// TIA Portal V15.1 export
// export: Created 2024-05-17T05:38:58.758149Z, ExportSetting WithDefaults, DisplayName Totally Integrated Automation Portal, DisplayVersion V15.1 Update 5, DisplayName TIA Portal Openness, DisplayVersion V15.1 Update 5, DisplayName SINAMICS Startdrive Advanced, DisplayVersion V15.1, DisplayName G130, G150, S120, S150, SINAMICS MV, S210, DisplayVersion V15.1, DisplayName G110M, G120, G120C, G120D, G120P, DisplayVersion V15.1, DisplayName STEP 7 Professional, DisplayVersion V15.1 Update 5, DisplayName STEP 7 Safety, DisplayVersion V15.1, DisplayName WinCC Professional, DisplayVersion V15.1 Update 5, DisplayName SIMATIC Visualization Architect, DisplayVersion V15.1
FUNCTION "209230ZS01PNIODiag" : Void   // FC424, FBD
TITLE = 209230ZS01PNIODiag
{ S7_Optimized_Access := 'FALSE' }
AUTHOR : JS
NAME : Mot001
VERSION : 0.1
// stored: AutoNumber false, IsIECCheckEnabled false, SetENOAutomatically False, UDAEnableTagReadback false
   VAR_OUTPUT
      O_AlarmA : Bool;   // Alarm A
      O_AlarmB : Bool;   // Alarm B
      O_AlarmC : Bool;   // Alarm C
      O_AlarmD : Bool;   // Alarm D
      O_AlarmABCondition : Bool;   // Alarms resetable
      H_IAnim : Word;   // Animation bits to Icon in WinCC
   END_VAR
   VAR_TEMP   // added for the SCL form of the ladder/FBD networks
      _w1 : Bool;
   END_VAR
BEGIN

REGION Network 1: **** --------------------- ET200sp I/O --------------------- ****
END_REGION

REGION Network 2: **** 3 - Communication - Devices **** 209230AS10-JW60 - ET200sp I/O - Busnode 230AS10 - node 60
   // Profinet device don't exist - ET200sp I/O - Busnode 230AS10 - node 60
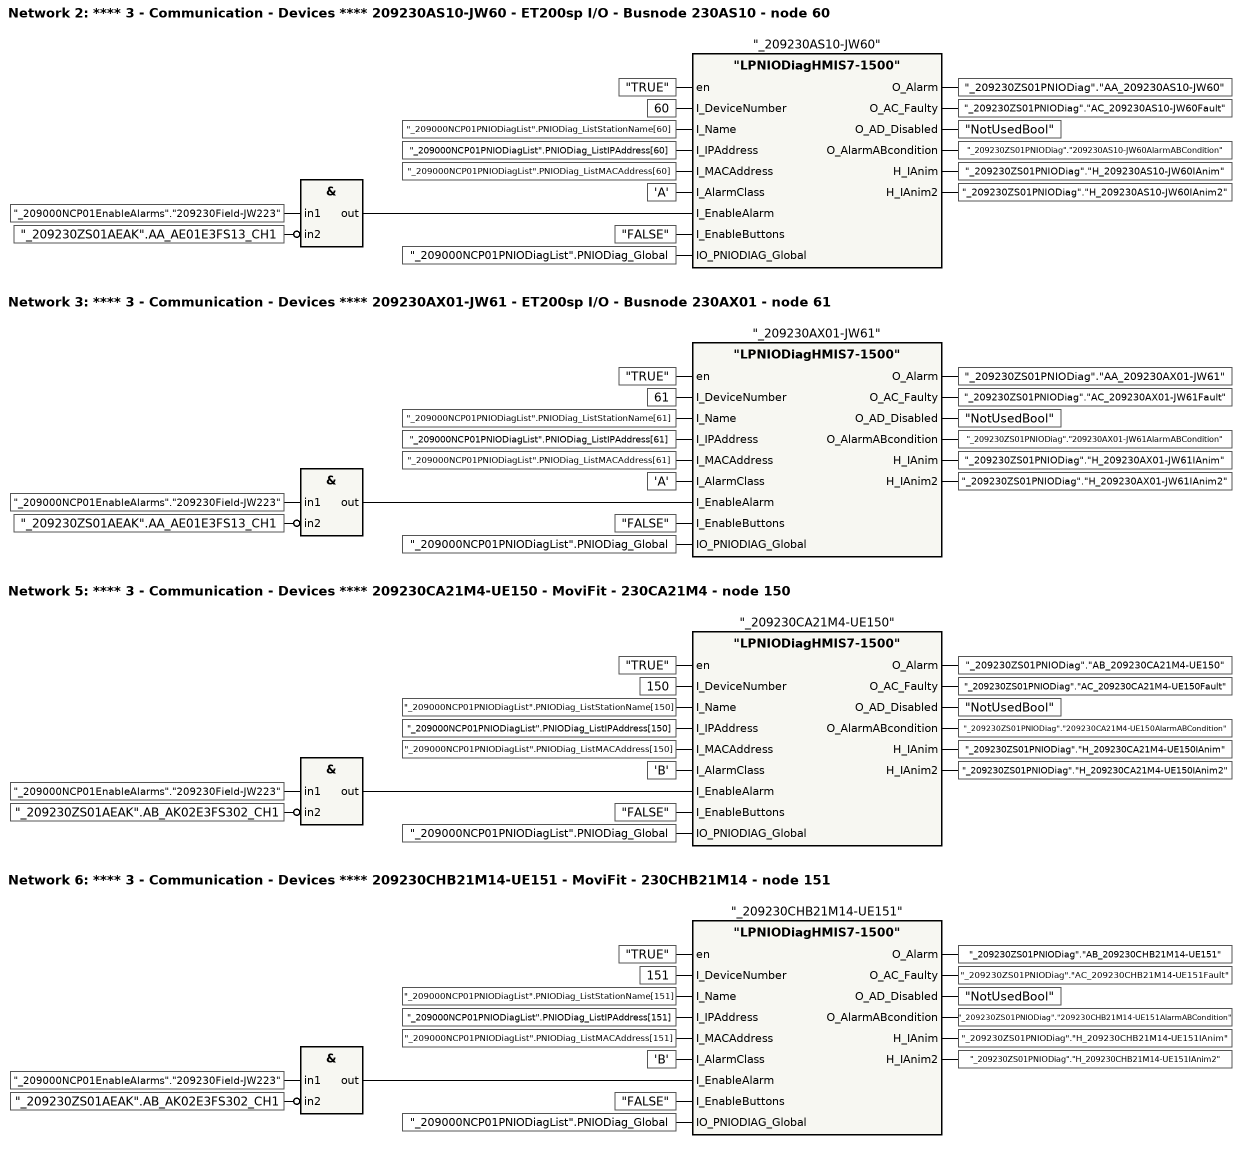
   IF "TRUE" THEN
       "_209230AS10-JW60"(I_DeviceNumber := 60,   // "LPNIODiagHMIS7-1500"
                          I_Name := "_209000NCP01PNIODiagList".PNIODiag_ListStationName[60],
                          I_IPAddress := "_209000NCP01PNIODiagList".PNIODiag_ListIPAddress[60],
                          I_MACAddress := "_209000NCP01PNIODiagList".PNIODiag_ListMACAddress[60],
                          I_AlarmClass := 'A',
                          I_EnableAlarm := "_209000NCP01EnableAlarms"."209230Field-JW223" AND NOT "_209230ZS01AEAK".AA_AE01E3FS13_CH1,
                          I_EnableButtons := "FALSE",
                          IO_PNIODIAG_Global := "_209000NCP01PNIODiagList".PNIODiag_Global,
                          O_Alarm => "_209230ZS01PNIODiag"."AA_209230AS10-JW60",
                          O_AC_Faulty => "_209230ZS01PNIODiag"."AC_209230AS10-JW60Fault",
                          O_AD_Disabled => "NotUsedBool",
                          O_AlarmABcondition => "_209230ZS01PNIODiag"."209230AS10-JW60AlarmABCondition",
                          H_IAnim => "_209230ZS01PNIODiag"."H_209230AS10-JW60IAnim",
                          H_IAnim2 => "_209230ZS01PNIODiag"."H_209230AS10-JW60IAnim2");
   END_IF;
END_REGION

REGION Network 3: **** 3 - Communication - Devices **** 209230AX01-JW61 - ET200sp I/O - Busnode 230AX01 - node 61
   // Profinet device don't exist - ET200sp I/O - Busnode 230AX01 - node 61
   IF "TRUE" THEN
       "_209230AX01-JW61"(I_DeviceNumber := 61,   // "LPNIODiagHMIS7-1500"
                          I_Name := "_209000NCP01PNIODiagList".PNIODiag_ListStationName[61],
                          I_IPAddress := "_209000NCP01PNIODiagList".PNIODiag_ListIPAddress[61],
                          I_MACAddress := "_209000NCP01PNIODiagList".PNIODiag_ListMACAddress[61],
                          I_AlarmClass := 'A',
                          I_EnableAlarm := "_209000NCP01EnableAlarms"."209230Field-JW223" AND NOT "_209230ZS01AEAK".AA_AE01E3FS13_CH1,
                          I_EnableButtons := "FALSE",
                          IO_PNIODIAG_Global := "_209000NCP01PNIODiagList".PNIODiag_Global,
                          O_Alarm => "_209230ZS01PNIODiag"."AA_209230AX01-JW61",
                          O_AC_Faulty => "_209230ZS01PNIODiag"."AC_209230AX01-JW61Fault",
                          O_AD_Disabled => "NotUsedBool",
                          O_AlarmABcondition => "_209230ZS01PNIODiag"."209230AX01-JW61AlarmABCondition",
                          H_IAnim => "_209230ZS01PNIODiag"."H_209230AX01-JW61IAnim",
                          H_IAnim2 => "_209230ZS01PNIODiag"."H_209230AX01-JW61IAnim2");
   END_IF;
END_REGION

REGION Network 4: **** --------------------- Drive --------------------- ****
END_REGION

REGION Network 5: **** 3 - Communication - Devices **** 209230CA21M4-UE150 - MoviFit - 230CA21M4 - node 150
   // Profinet device don't exist - MoviFit - 230CA21M4 - node 150
   IF "TRUE" THEN
       "_209230CA21M4-UE150"(I_DeviceNumber := 150,   // "LPNIODiagHMIS7-1500"
                             I_Name := "_209000NCP01PNIODiagList".PNIODiag_ListStationName[150],
                             I_IPAddress := "_209000NCP01PNIODiagList".PNIODiag_ListIPAddress[150],
                             I_MACAddress := "_209000NCP01PNIODiagList".PNIODiag_ListMACAddress[150],
                             I_AlarmClass := 'B',
                             I_EnableAlarm := "_209000NCP01EnableAlarms"."209230Field-JW223" AND NOT "_209230ZS01AEAK".AB_AK02E3FS302_CH1,
                             I_EnableButtons := "FALSE",
                             IO_PNIODIAG_Global := "_209000NCP01PNIODiagList".PNIODiag_Global,
                             O_Alarm => "_209230ZS01PNIODiag"."AB_209230CA21M4-UE150",
                             O_AC_Faulty => "_209230ZS01PNIODiag"."AC_209230CA21M4-UE150Fault",
                             O_AD_Disabled => "NotUsedBool",
                             O_AlarmABcondition => "_209230ZS01PNIODiag"."209230CA21M4-UE150AlarmABCondition",
                             H_IAnim => "_209230ZS01PNIODiag"."H_209230CA21M4-UE150IAnim",
                             H_IAnim2 => "_209230ZS01PNIODiag"."H_209230CA21M4-UE150IAnim2");
   END_IF;
END_REGION

REGION Network 6: **** 3 - Communication - Devices **** 209230CHB21M14-UE151 - MoviFit - 230CHB21M14 - node 151
   // Profinet device don't exist - MoviFit - 230CHB21M14 - node 151
   IF "TRUE" THEN
       "_209230CHB21M14-UE151"(I_DeviceNumber := 151,   // "LPNIODiagHMIS7-1500"
                               I_Name := "_209000NCP01PNIODiagList".PNIODiag_ListStationName[151],
                               I_IPAddress := "_209000NCP01PNIODiagList".PNIODiag_ListIPAddress[151],
                               I_MACAddress := "_209000NCP01PNIODiagList".PNIODiag_ListMACAddress[151],
                               I_AlarmClass := 'B',
                               I_EnableAlarm := "_209000NCP01EnableAlarms"."209230Field-JW223" AND NOT "_209230ZS01AEAK".AB_AK02E3FS302_CH1,
                               I_EnableButtons := "FALSE",
                               IO_PNIODIAG_Global := "_209000NCP01PNIODiagList".PNIODiag_Global,
                               O_Alarm => "_209230ZS01PNIODiag"."AB_209230CHB21M14-UE151",
                               O_AC_Faulty => "_209230ZS01PNIODiag"."AC_209230CHB21M14-UE151Fault",
                               O_AD_Disabled => "NotUsedBool",
                               O_AlarmABcondition => "_209230ZS01PNIODiag"."209230CHB21M14-UE151AlarmABCondition",
                               H_IAnim => "_209230ZS01PNIODiag"."H_209230CHB21M14-UE151IAnim",
                               H_IAnim2 => "_209230ZS01PNIODiag"."H_209230CHB21M14-UE151IAnim2");
   END_IF;
END_REGION

REGION Network 7: **** 3 - Communication - Devices **** 209230CHB22M14-UE152 - MoviFit - 230CHB22M14 - node 152
   // Profinet device don't exist - MoviFit - 230CHB22M14 - node 152
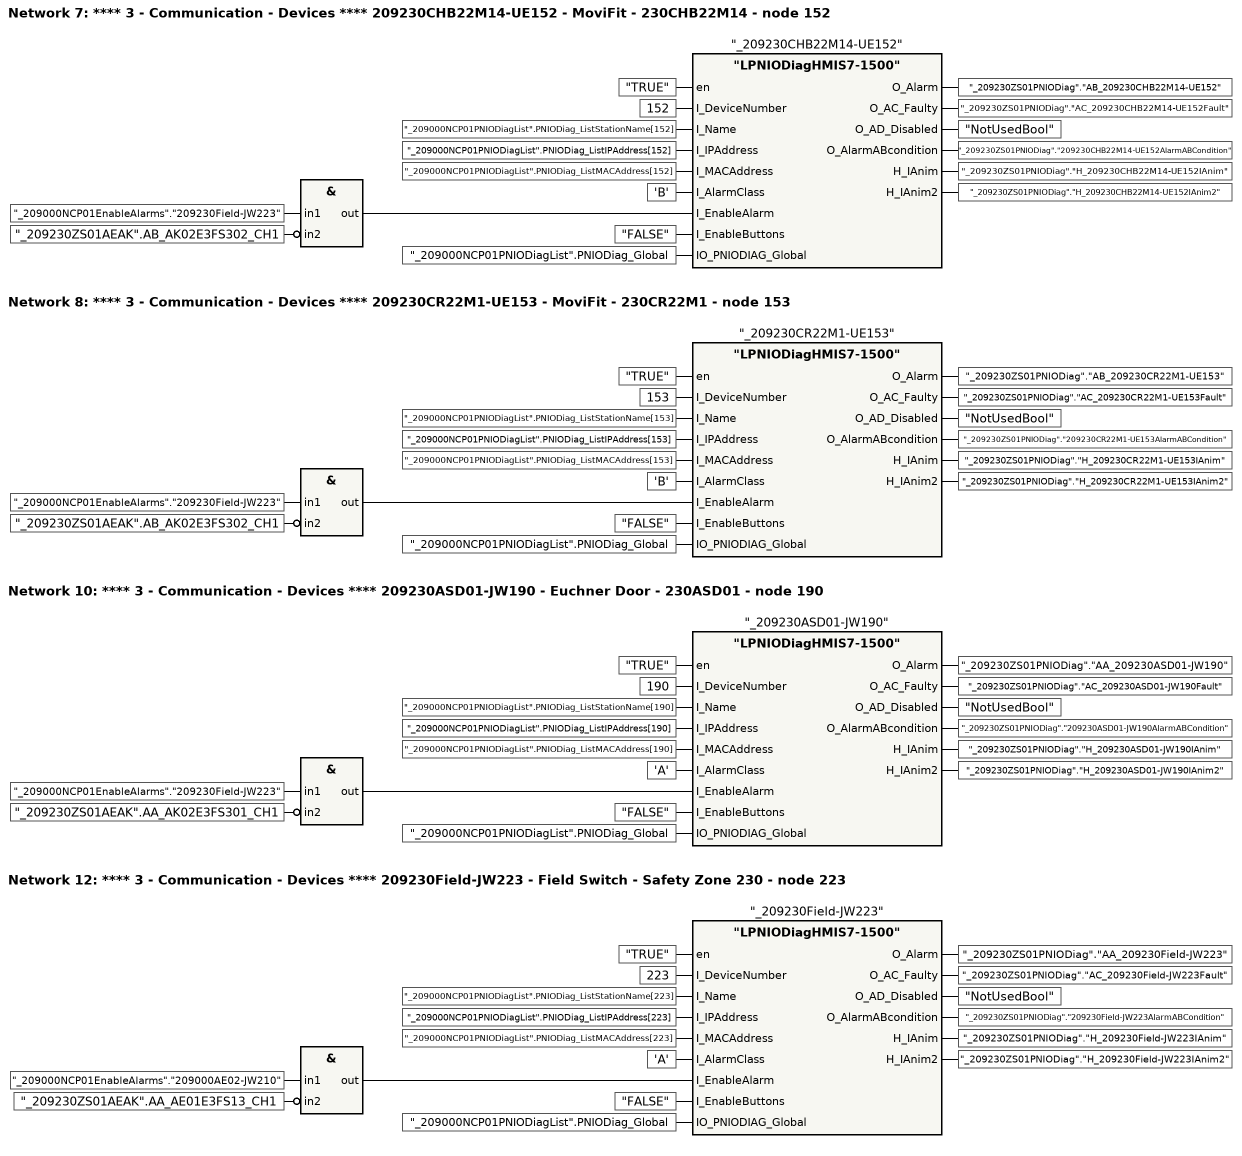
   IF "TRUE" THEN
       "_209230CHB22M14-UE152"(I_DeviceNumber := 152,   // "LPNIODiagHMIS7-1500"
                               I_Name := "_209000NCP01PNIODiagList".PNIODiag_ListStationName[152],
                               I_IPAddress := "_209000NCP01PNIODiagList".PNIODiag_ListIPAddress[152],
                               I_MACAddress := "_209000NCP01PNIODiagList".PNIODiag_ListMACAddress[152],
                               I_AlarmClass := 'B',
                               I_EnableAlarm := "_209000NCP01EnableAlarms"."209230Field-JW223" AND NOT "_209230ZS01AEAK".AB_AK02E3FS302_CH1,
                               I_EnableButtons := "FALSE",
                               IO_PNIODIAG_Global := "_209000NCP01PNIODiagList".PNIODiag_Global,
                               O_Alarm => "_209230ZS01PNIODiag"."AB_209230CHB22M14-UE152",
                               O_AC_Faulty => "_209230ZS01PNIODiag"."AC_209230CHB22M14-UE152Fault",
                               O_AD_Disabled => "NotUsedBool",
                               O_AlarmABcondition => "_209230ZS01PNIODiag"."209230CHB22M14-UE152AlarmABCondition",
                               H_IAnim => "_209230ZS01PNIODiag"."H_209230CHB22M14-UE152IAnim",
                               H_IAnim2 => "_209230ZS01PNIODiag"."H_209230CHB22M14-UE152IAnim2");
   END_IF;
END_REGION

REGION Network 8: **** 3 - Communication - Devices **** 209230CR22M1-UE153 - MoviFit - 230CR22M1 - node 153
   // Profinet device don't exist - MoviFit - 230CR22M1 - node 153
   IF "TRUE" THEN
       "_209230CR22M1-UE153"(I_DeviceNumber := 153,   // "LPNIODiagHMIS7-1500"
                             I_Name := "_209000NCP01PNIODiagList".PNIODiag_ListStationName[153],
                             I_IPAddress := "_209000NCP01PNIODiagList".PNIODiag_ListIPAddress[153],
                             I_MACAddress := "_209000NCP01PNIODiagList".PNIODiag_ListMACAddress[153],
                             I_AlarmClass := 'B',
                             I_EnableAlarm := "_209000NCP01EnableAlarms"."209230Field-JW223" AND NOT "_209230ZS01AEAK".AB_AK02E3FS302_CH1,
                             I_EnableButtons := "FALSE",
                             IO_PNIODIAG_Global := "_209000NCP01PNIODiagList".PNIODiag_Global,
                             O_Alarm => "_209230ZS01PNIODiag"."AB_209230CR22M1-UE153",
                             O_AC_Faulty => "_209230ZS01PNIODiag"."AC_209230CR22M1-UE153Fault",
                             O_AD_Disabled => "NotUsedBool",
                             O_AlarmABcondition => "_209230ZS01PNIODiag"."209230CR22M1-UE153AlarmABCondition",
                             H_IAnim => "_209230ZS01PNIODiag"."H_209230CR22M1-UE153IAnim",
                             H_IAnim2 => "_209230ZS01PNIODiag"."H_209230CR22M1-UE153IAnim2");
   END_IF;
END_REGION

REGION Network 9: **** --------------------- Euchner Door --------------------- ****
END_REGION

REGION Network 10: **** 3 - Communication - Devices **** 209230ASD01-JW190 - Euchner Door - 230ASD01 - node 190
   // Profinet device don't exist - Euchner Door - 230ASD01 - node 190
   IF "TRUE" THEN
       "_209230ASD01-JW190"(I_DeviceNumber := 190,   // "LPNIODiagHMIS7-1500"
                            I_Name := "_209000NCP01PNIODiagList".PNIODiag_ListStationName[190],
                            I_IPAddress := "_209000NCP01PNIODiagList".PNIODiag_ListIPAddress[190],
                            I_MACAddress := "_209000NCP01PNIODiagList".PNIODiag_ListMACAddress[190],
                            I_AlarmClass := 'A',
                            I_EnableAlarm := "_209000NCP01EnableAlarms"."209230Field-JW223" AND NOT "_209230ZS01AEAK".AA_AK02E3FS301_CH1,
                            I_EnableButtons := "FALSE",
                            IO_PNIODIAG_Global := "_209000NCP01PNIODiagList".PNIODiag_Global,
                            O_Alarm => "_209230ZS01PNIODiag"."AA_209230ASD01-JW190",
                            O_AC_Faulty => "_209230ZS01PNIODiag"."AC_209230ASD01-JW190Fault",
                            O_AD_Disabled => "NotUsedBool",
                            O_AlarmABcondition => "_209230ZS01PNIODiag"."209230ASD01-JW190AlarmABCondition",
                            H_IAnim => "_209230ZS01PNIODiag"."H_209230ASD01-JW190IAnim",
                            H_IAnim2 => "_209230ZS01PNIODiag"."H_209230ASD01-JW190IAnim2");
   END_IF;
END_REGION

REGION Network 11: **** --------------------- Field Switch --------------------- ****
END_REGION

REGION Network 12: **** 3 - Communication - Devices **** 209230Field-JW223 - Field Switch - Safety Zone 230 - node 223
   // Profinet device don't exist - Field Switch - Safety Zone 230 - node 223
   IF "TRUE" THEN
       "_209230Field-JW223"(I_DeviceNumber := 223,   // "LPNIODiagHMIS7-1500"
                            I_Name := "_209000NCP01PNIODiagList".PNIODiag_ListStationName[223],
                            I_IPAddress := "_209000NCP01PNIODiagList".PNIODiag_ListIPAddress[223],
                            I_MACAddress := "_209000NCP01PNIODiagList".PNIODiag_ListMACAddress[223],
                            I_AlarmClass := 'A',
                            I_EnableAlarm := "_209000NCP01EnableAlarms"."209000AE02-JW210" AND NOT "_209230ZS01AEAK".AA_AE01E3FS13_CH1,
                            I_EnableButtons := "FALSE",
                            IO_PNIODIAG_Global := "_209000NCP01PNIODiagList".PNIODiag_Global,
                            O_Alarm => "_209230ZS01PNIODiag"."AA_209230Field-JW223",
                            O_AC_Faulty => "_209230ZS01PNIODiag"."AC_209230Field-JW223Fault",
                            O_AD_Disabled => "NotUsedBool",
                            O_AlarmABcondition => "_209230ZS01PNIODiag"."209230Field-JW223AlarmABCondition",
                            H_IAnim => "_209230ZS01PNIODiag"."H_209230Field-JW223IAnim",
                            H_IAnim2 => "_209230ZS01PNIODiag"."H_209230Field-JW223IAnim2");
   END_IF;
END_REGION

REGION Network 13: **** -------------------------------------------------- ****
END_REGION

REGION Network 14: **** 4.6 - Machine Status - Indications **** Icon animation
   // Icon animation
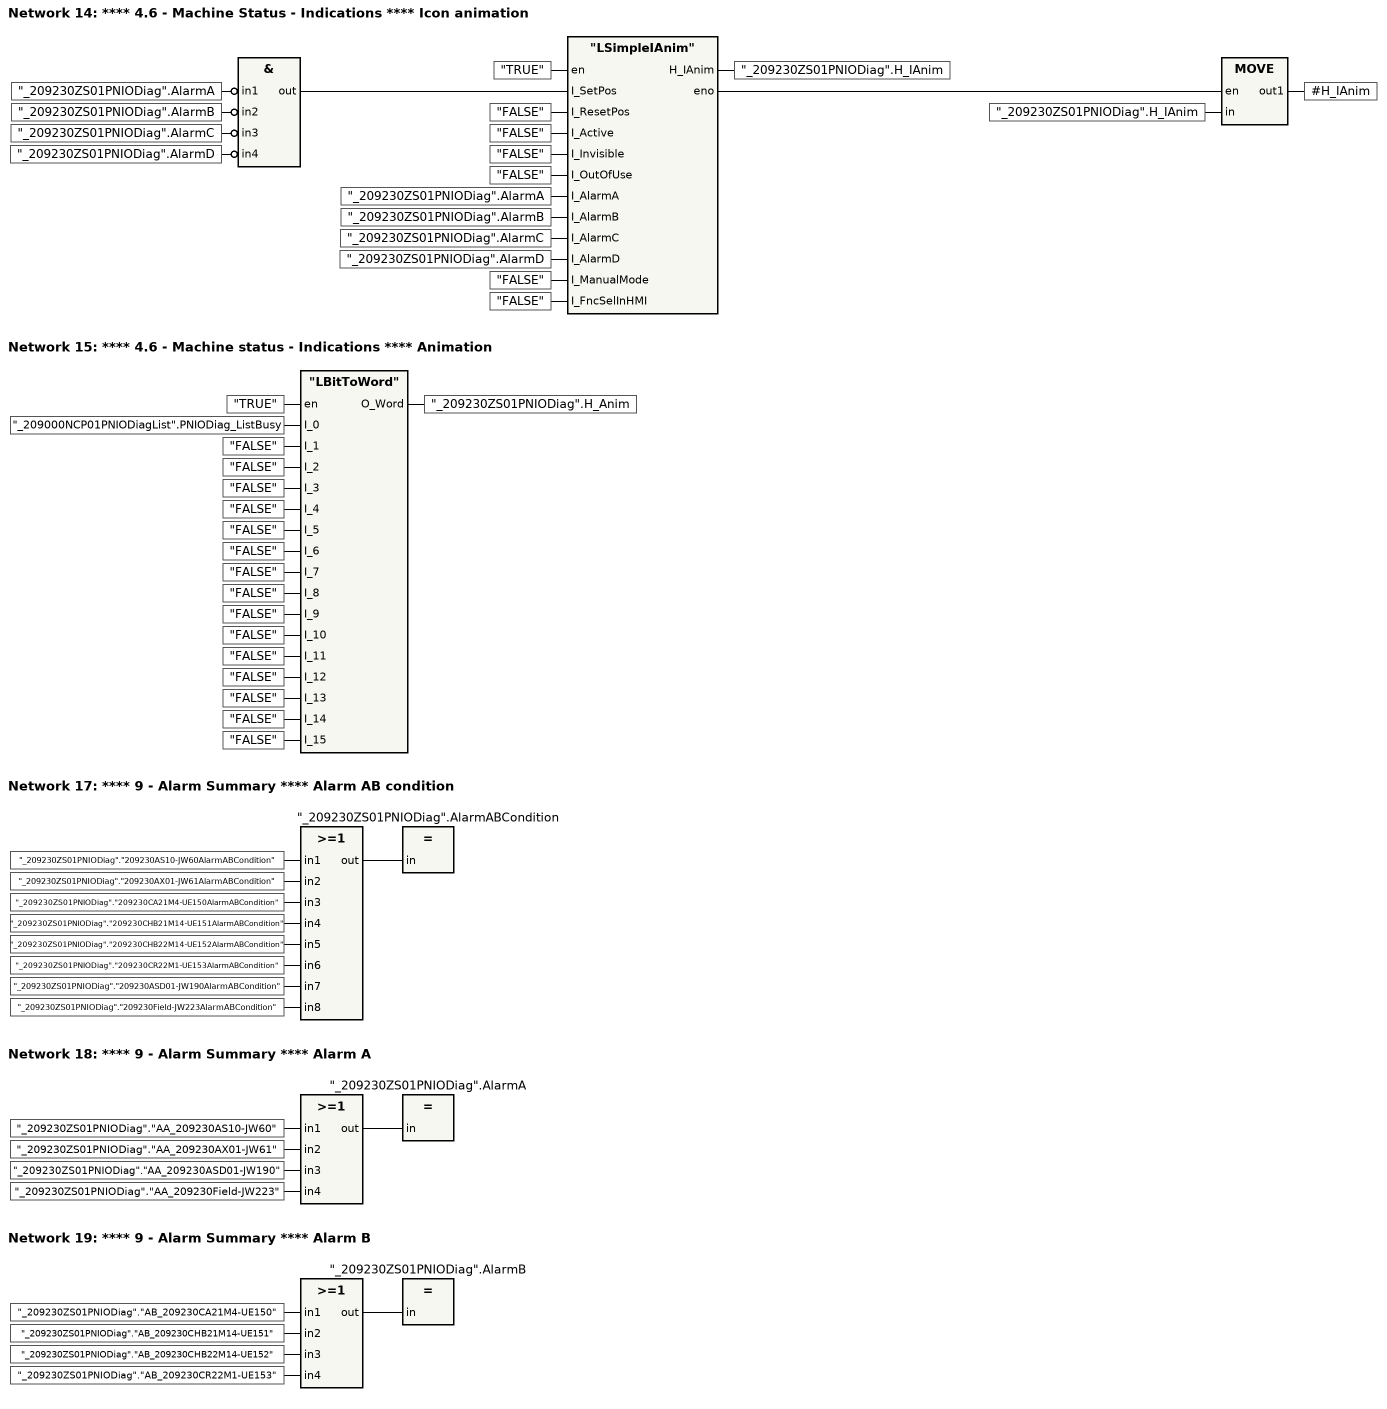
   "LSimpleIAnim"(EN := "TRUE",
                  I_SetPos := NOT "_209230ZS01PNIODiag".AlarmA AND NOT "_209230ZS01PNIODiag".AlarmB AND NOT "_209230ZS01PNIODiag".AlarmC AND NOT "_209230ZS01PNIODiag".AlarmD,
                  I_ResetPos := "FALSE",
                  I_Active := "FALSE",
                  I_Invisible := "FALSE",
                  I_OutOfUse := "FALSE",
                  I_AlarmA := "_209230ZS01PNIODiag".AlarmA,
                  I_AlarmB := "_209230ZS01PNIODiag".AlarmB,
                  I_AlarmC := "_209230ZS01PNIODiag".AlarmC,
                  I_AlarmD := "_209230ZS01PNIODiag".AlarmD,
                  I_ManualMode := "FALSE",
                  I_FncSelInHMI := "FALSE",
                  H_IAnim => "_209230ZS01PNIODiag".H_IAnim,
                  ENO => #_w1);
   IF #_w1 THEN #H_IAnim := "_209230ZS01PNIODiag".H_IAnim; END_IF;
END_REGION

REGION Network 15: **** 4.6 - Machine status - Indications **** Animation
   // Animation
   IF "TRUE" THEN
       "LBitToWord"(I_0 := "_209000NCP01PNIODiagList".PNIODiag_ListBusy,
                    I_1 := "FALSE",
                    I_2 := "FALSE",
                    I_3 := "FALSE",
                    I_4 := "FALSE",
                    I_5 := "FALSE",
                    I_6 := "FALSE",
                    I_7 := "FALSE",
                    I_8 := "FALSE",
                    I_9 := "FALSE",
                    I_10 := "FALSE",
                    I_11 := "FALSE",
                    I_12 := "FALSE",
                    I_13 := "FALSE",
                    I_14 := "FALSE",
                    I_15 := "FALSE",
                    O_Word => "_209230ZS01PNIODiag".H_Anim);
   END_IF;
END_REGION

NETWORK
TITLE = **** 4.6 - Machine Status - Indications **** Animation DB number
// DB number
      OPN   "_209230ZS01PNIODiag";
      L     DBNO;
      T     "_209230ZS01PNIODiag".H_DBnr;

REGION Network 17: **** 9 - Alarm Summary **** Alarm AB condition
   // Summary of Alarm AB condition
   "_209230ZS01PNIODiag".AlarmABCondition := "_209230ZS01PNIODiag"."209230AS10-JW60AlarmABCondition" OR "_209230ZS01PNIODiag"."209230AX01-JW61AlarmABCondition" OR "_209230ZS01PNIODiag"."209230CA21M4-UE150AlarmABCondition" OR "_209230ZS01PNIODiag"."209230CHB21M14-UE151AlarmABCondition" OR "_209230ZS01PNIODiag"."209230CHB22M14-UE152AlarmABCondition" OR "_209230ZS01PNIODiag"."209230CR22M1-UE153AlarmABCondition" OR "_209230ZS01PNIODiag"."209230ASD01-JW190AlarmABCondition" OR "_209230ZS01PNIODiag"."209230Field-JW223AlarmABCondition";
END_REGION

REGION Network 18: **** 9 - Alarm Summary **** Alarm A
   // Summary of alarms A
   "_209230ZS01PNIODiag".AlarmA := "_209230ZS01PNIODiag"."AA_209230AS10-JW60" OR "_209230ZS01PNIODiag"."AA_209230AX01-JW61" OR "_209230ZS01PNIODiag"."AA_209230ASD01-JW190" OR "_209230ZS01PNIODiag"."AA_209230Field-JW223";
END_REGION

REGION Network 19: **** 9 - Alarm Summary **** Alarm B
   // Summary of alarms B
   "_209230ZS01PNIODiag".AlarmB := "_209230ZS01PNIODiag"."AB_209230CA21M4-UE150" OR "_209230ZS01PNIODiag"."AB_209230CHB21M14-UE151" OR "_209230ZS01PNIODiag"."AB_209230CHB22M14-UE152" OR "_209230ZS01PNIODiag"."AB_209230CR22M1-UE153";
END_REGION

REGION Network 20: **** 9 - Alarm Summary **** Alarm C
   // Summary of alarms C
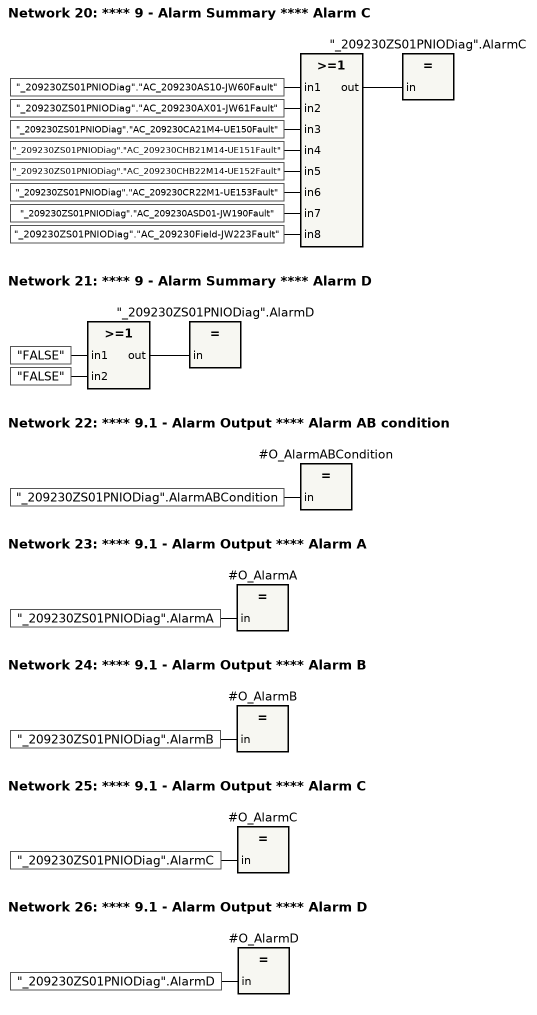
   "_209230ZS01PNIODiag".AlarmC := "_209230ZS01PNIODiag"."AC_209230AS10-JW60Fault" OR "_209230ZS01PNIODiag"."AC_209230AX01-JW61Fault" OR "_209230ZS01PNIODiag"."AC_209230CA21M4-UE150Fault" OR "_209230ZS01PNIODiag"."AC_209230CHB21M14-UE151Fault" OR "_209230ZS01PNIODiag"."AC_209230CHB22M14-UE152Fault" OR "_209230ZS01PNIODiag"."AC_209230CR22M1-UE153Fault" OR "_209230ZS01PNIODiag"."AC_209230ASD01-JW190Fault" OR "_209230ZS01PNIODiag"."AC_209230Field-JW223Fault";
END_REGION

REGION Network 21: **** 9 - Alarm Summary **** Alarm D
   // Summary of alarms D
   "_209230ZS01PNIODiag".AlarmD := "FALSE" OR "FALSE";
END_REGION

REGION Network 22: **** 9.1 - Alarm Output **** Alarm AB condition
   // Alarm AB condition
   #O_AlarmABCondition := "_209230ZS01PNIODiag".AlarmABCondition;
END_REGION

REGION Network 23: **** 9.1 - Alarm Output **** Alarm A
   // Output Alarm A
   #O_AlarmA := "_209230ZS01PNIODiag".AlarmA;
END_REGION

REGION Network 24: **** 9.1 - Alarm Output **** Alarm B
   // Output Alarm B
   #O_AlarmB := "_209230ZS01PNIODiag".AlarmB;
END_REGION

REGION Network 25: **** 9.1 - Alarm Output **** Alarm C
   // Output Alarm A
   #O_AlarmC := "_209230ZS01PNIODiag".AlarmC;
END_REGION

REGION Network 26: **** 9.1 - Alarm Output **** Alarm D
   // Output Alarm D
   #O_AlarmD := "_209230ZS01PNIODiag".AlarmD;
END_REGION

REGION Network 27: **** 9.2 - Alarm DWord**** Alarm To DWord
   // Alarm Word
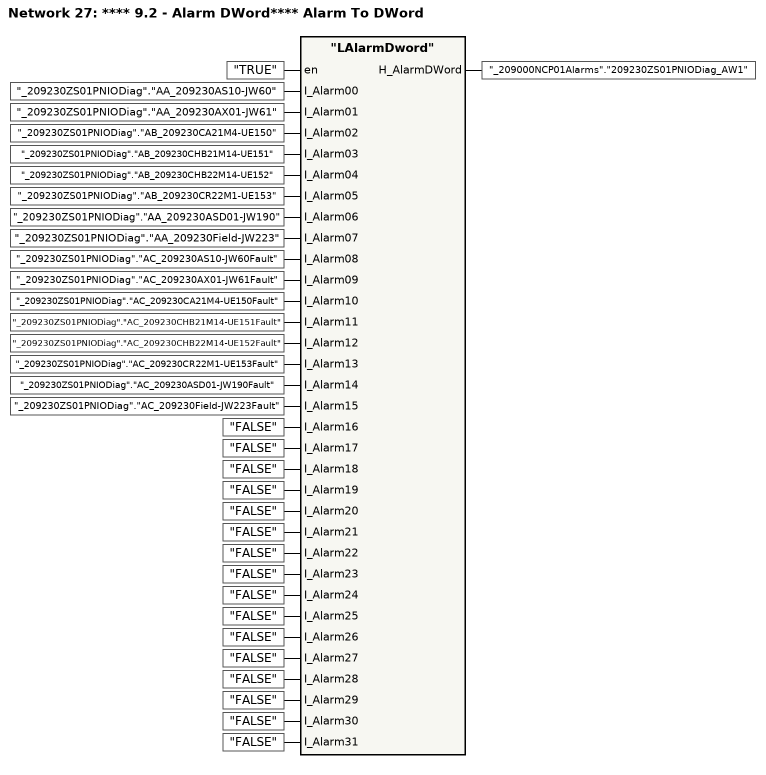
   IF "TRUE" THEN
       "LAlarmDword"(I_Alarm00 := "_209230ZS01PNIODiag"."AA_209230AS10-JW60",
                     I_Alarm01 := "_209230ZS01PNIODiag"."AA_209230AX01-JW61",
                     I_Alarm02 := "_209230ZS01PNIODiag"."AB_209230CA21M4-UE150",
                     I_Alarm03 := "_209230ZS01PNIODiag"."AB_209230CHB21M14-UE151",
                     I_Alarm04 := "_209230ZS01PNIODiag"."AB_209230CHB22M14-UE152",
                     I_Alarm05 := "_209230ZS01PNIODiag"."AB_209230CR22M1-UE153",
                     I_Alarm06 := "_209230ZS01PNIODiag"."AA_209230ASD01-JW190",
                     I_Alarm07 := "_209230ZS01PNIODiag"."AA_209230Field-JW223",
                     I_Alarm08 := "_209230ZS01PNIODiag"."AC_209230AS10-JW60Fault",
                     I_Alarm09 := "_209230ZS01PNIODiag"."AC_209230AX01-JW61Fault",
                     I_Alarm10 := "_209230ZS01PNIODiag"."AC_209230CA21M4-UE150Fault",
                     I_Alarm11 := "_209230ZS01PNIODiag"."AC_209230CHB21M14-UE151Fault",
                     I_Alarm12 := "_209230ZS01PNIODiag"."AC_209230CHB22M14-UE152Fault",
                     I_Alarm13 := "_209230ZS01PNIODiag"."AC_209230CR22M1-UE153Fault",
                     I_Alarm14 := "_209230ZS01PNIODiag"."AC_209230ASD01-JW190Fault",
                     I_Alarm15 := "_209230ZS01PNIODiag"."AC_209230Field-JW223Fault",
                     I_Alarm16 := "FALSE",
                     I_Alarm17 := "FALSE",
                     I_Alarm18 := "FALSE",
                     I_Alarm19 := "FALSE",
                     I_Alarm20 := "FALSE",
                     I_Alarm21 := "FALSE",
                     I_Alarm22 := "FALSE",
                     I_Alarm23 := "FALSE",
                     I_Alarm24 := "FALSE",
                     I_Alarm25 := "FALSE",
                     I_Alarm26 := "FALSE",
                     I_Alarm27 := "FALSE",
                     I_Alarm28 := "FALSE",
                     I_Alarm29 := "FALSE",
                     I_Alarm30 := "FALSE",
                     I_Alarm31 := "FALSE",
                     H_AlarmDWord => "_209000NCP01Alarms"."209230ZS01PNIODiag_AW1");
   END_IF;
END_REGION
END_FUNCTION
